(* IEC 61131-3 sources: CodesysTest/alpha/export/Pro18_1174_Win10.dev/Plc Logic/Application/Motors/Applied Motion/DataHandlers/FB_StepServoCommands.pou/FeedToLength.prop, 1 file *)

(* ---- Set.pm.st ---- *)
(*#-#-#-#-#-#-#-#-#-#---Declaration---#-#-#-#-#-#-#-#-#-#-#-#-#*)

VAR
END_VAR
(*#-#-#-#-#-#-#-#-#-#---Implementation---#-#-#-#-#-#-#-#-#-#-#-#-#*)

commandSent := FALSE;
_feedToLength := FeedToLength;
